FUNCTION_BLOCK Basic (* Basic FB with empty ECC *)
  (* Standard: 61499-2 *)
  (* Version 1.0, 2016-05-26, AZ, fortiss GmbH *)
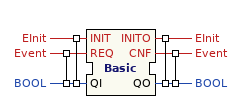
  EVENT_INPUT
    INIT : EInit WITH QI; (* Initialization Request *)
    REQ WITH QI; (* Normal Execution Request *)
  END_EVENT
  EVENT_OUTPUT
    INITO : EInit WITH QO; (* Initialization Confirm *)
    CNF WITH QO; (* Execution Confirmation *)
  END_EVENT
  VAR_INPUT
    QI : BOOL; (* Input event qualifier *)
  END_VAR
  VAR_OUTPUT
    QO : BOOL; (* Output event qualifier *)
  END_VAR
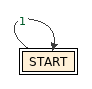
  EC_STATES
    START; (* Initial State *)
  END_STATES
  EC_TRANSITIONS
    START TO START := 1; (* pls modify this! *)
  END_TRANSITIONS
END_FUNCTION_BLOCK
